(* CODESYS project Mehatronika_seminarski.project
   Title: PMS_LV9_z1
   Version: 0.0.0.0
   Author: CA Simple

Project tree, tasks and I/O mapping:
  MyController : TM238LDD24DT, Schneider Electric, order no. TM238LDD24DT, version 4.0.1.28
      settings: OpcUa Enable = False
    application Application
      task MAST (cyclic, interval 20 ms, priority 15, watchdog 100 ms x 1) calls POU
      global variables GVL
      program POU [SFC]: Init_entry, Step4_entry, kafa0_active, kafa0_entry, Step1_entry, Step2_entry, kafa0_exit, caj1_active, kafa1_exit, kafa2_active, kafa2_exit, kafa1_active, caj2_active, caj1_exit, caj2_exit, caj0_entry, caj0_exit, caj0_active, kakao0_entry, kapucino0_entry, kakao0_exit, kapucino0_exit, kakao0_active, kapucino0_active, kakao1_active, kakao1_exit, kakao2_active, kakao2_exit, kapucino1_active, kapucino1_exit, kapucino3_active, kapucino3_exit, kapucino2_active, kapucino2_exit, kafa1_entry, kafa2_entry, caj1_entry, caj2_entry, kakao1_entry, kapucino1_entry, kakao2_entry, kapucino2_entry, kapucino3_entry, Init_active, preuzimanje_active_0, Init_exit, preuzimanje_exit
      Symbols
    Embedded Functions
      IO : IO, Schneider Electric, version 4.0.1.28
          input  Application.polaKM : BOOL  // IW0.I0
          input  Application.jedanKM : BOOL  // IW0.I1
          input  Application.dvaKM : BOOL  // IW0.I2
          input  Application.kafa : BOOL  // IW0.I3
          input  Application.caj : BOOL  // IW0.I4
          input  Application.kakao : BOOL  // IW0.I5
          input  Application.kapucino : BOOL  // IW0.I6
          output Application.voda : BOOL  // QW0.Q0
          output Application.posuda1 : BOOL  // QW0.Q1
          output Application.posuda2 : BOOL  // QW0.Q2
          output Application.posuda3 : BOOL  // QW0.Q3
          output Application.posuda4 : BOOL  // QW0.Q4
          output Application.posuda5 : BOOL  // QW0.Q5
          unmapped channels: IW0, QW0
      HSC : HSC, Schneider Electric, version 4.0.1.28
      PTO_PWM : PTO_PWM, Schneider Electric, version 4.0.1.28
    Serial Line
      SoMachine_Network_Manager : SoMachine-Network Manager, Schneider Electric, version 4.0.0.2
  HMIS5T : HMIS5T, Schneider Electric, order no. HMIS5T, version 3.5.3.54
    HMI Application
    COM1
      SoMachine_Network_Manager1 : SoMachine-Network Manager, Schneider Electric, version 4.0.0.2
    Ethernet
      SoMachine_Network_Manager2 : SoMachine-Network Manager, Schneider Electric, version 4.0.0.2
    USB
      SoMachine_Network_Manager3 : SoMachine-Network Manager, Schneider Electric, version 4.0.0.2
  Vijeo Designer Project Container Data
  Vijeo Designer Project Container
*)

// MyController/Application/GVL
VAR_GLOBAL
END_VAR
VAR_GLOBAL
	petKM: BOOL;
	dvaKM: BOOL;
	jedanKM: BOOL;
	polaKM: BOOL;
	posuda5: BOOL;
	posuda4: BOOL;
	posuda3: BOOL;
	posuda2: BOOL;
	posuda1: BOOL;
	voda: BOOL;
	kapucino: BOOL;
	kakao: BOOL;
	caj: BOOL;
	kafa: BOOL;
	iznos: REAL := 0;
	kafa_iznos: BOOL;
	caj_iznos: BOOL;
	kakao_iznos: BOOL;
	kapucino_iznos: BOOL;
	kafa_gotova: BOOL;
	caj_gotov: BOOL;
	kakao_gotov: BOOL;
	kapucino_gotov: BOOL;
	kafa_u_proizvodnji: BOOL;
	caj_u_proizvodnji: BOOL;
	kakao_u_proizvodnji: BOOL;
	kapucino_u_proizvodnji: BOOL;
	proizvod_pokupljen: BOOL;
END_VAR

// MyController/Application/POU
PROGRAM POU
VAR
	okidac_posuda5: BOOL;
	okidac_posuda4: BOOL;
	okidac_posuda3: BOOL;
	okidac_posuda2: BOOL;
	okidac_posuda1: BOOL;
	okidac_voda: BOOL;
	posuda5_timer: TP;
	posuda5_f_trig: F_TRIG;
	posuda4_timer: TP;
	posuda4_f_trig: F_TRIG;
	posuda3_timer: TP;
	posuda3_f_trig: F_TRIG;
	posuda2_timer: TP;
	posuda2_f_trig: F_TRIG;
	posuda1_timer: TP;
	posuda1_f_trig: F_TRIG;
	voda_timer: TP;
	voda_f_trig: F_TRIG;
	pomocna: BOOL;
END_VAR

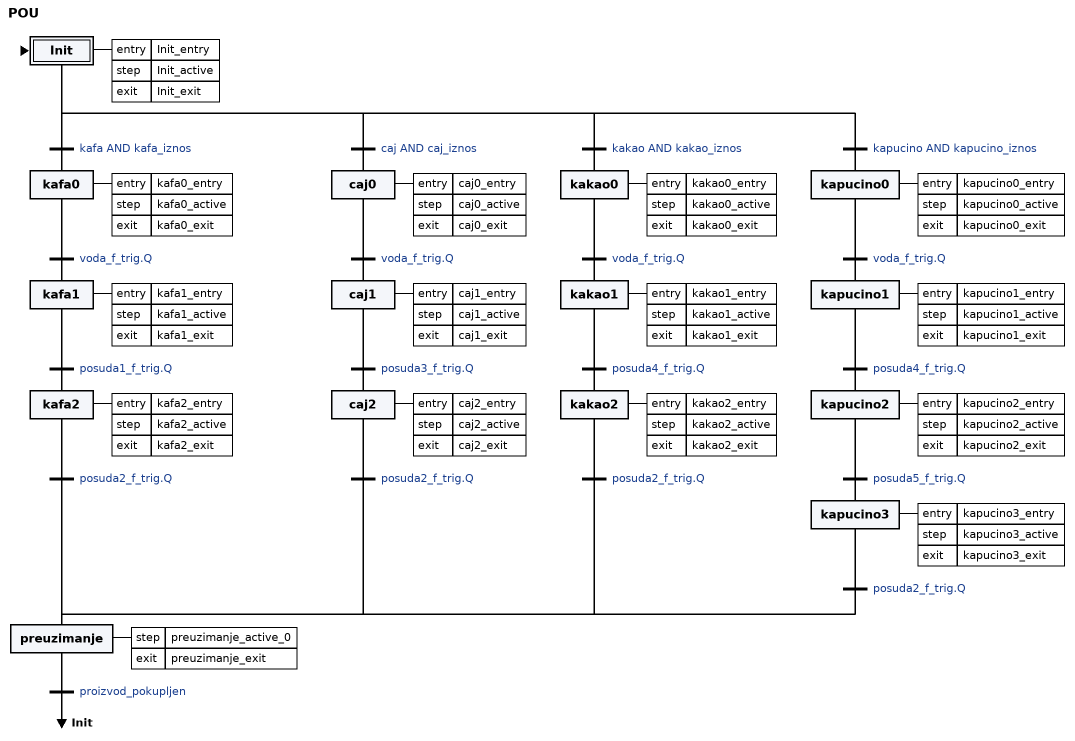
INITIAL_STEP Init:
    Init_entry(P1);  // entry action
    Init_active(N);  // step action
    Init_exit(P0);  // exit action
END_STEP
TRANSITION FROM Init TO kafa0
    := kafa AND kafa_iznos;
END_TRANSITION
STEP kafa0:
    kafa0_entry(P1);  // entry action
    kafa0_active(N);  // step action
    kafa0_exit(P0);  // exit action
END_STEP
TRANSITION FROM kafa0 TO kafa1
    := voda_f_trig.Q;
END_TRANSITION
STEP kafa1:
    kafa1_entry(P1);  // entry action
    kafa1_active(N);  // step action
    kafa1_exit(P0);  // exit action
END_STEP
TRANSITION FROM kafa1 TO kafa2
    := posuda1_f_trig.Q;
END_TRANSITION
STEP kafa2:
    kafa2_entry(P1);  // entry action
    kafa2_active(N);  // step action
    kafa2_exit(P0);  // exit action
END_STEP
TRANSITION FROM kafa2 TO preuzimanje
    := posuda2_f_trig.Q;
END_TRANSITION
TRANSITION FROM Init TO caj0
    := caj AND caj_iznos;
END_TRANSITION
STEP caj0:
    caj0_entry(P1);  // entry action
    caj0_active(N);  // step action
    caj0_exit(P0);  // exit action
END_STEP
TRANSITION FROM caj0 TO caj1
    := voda_f_trig.Q;
END_TRANSITION
STEP caj1:
    caj1_entry(P1);  // entry action
    caj1_active(N);  // step action
    caj1_exit(P0);  // exit action
END_STEP
TRANSITION FROM caj1 TO caj2
    := posuda3_f_trig.Q;
END_TRANSITION
STEP caj2:
    caj2_entry(P1);  // entry action
    caj2_active(N);  // step action
    caj2_exit(P0);  // exit action
END_STEP
TRANSITION FROM caj2 TO preuzimanje
    := posuda2_f_trig.Q;
END_TRANSITION
TRANSITION FROM Init TO kakao0
    := kakao AND kakao_iznos;
END_TRANSITION
STEP kakao0:
    kakao0_entry(P1);  // entry action
    kakao0_active(N);  // step action
    kakao0_exit(P0);  // exit action
END_STEP
TRANSITION FROM kakao0 TO kakao1
    := voda_f_trig.Q;
END_TRANSITION
STEP kakao1:
    kakao1_entry(P1);  // entry action
    kakao1_active(N);  // step action
    kakao1_exit(P0);  // exit action
END_STEP
TRANSITION FROM kakao1 TO kakao2
    := posuda4_f_trig.Q;
END_TRANSITION
STEP kakao2:
    kakao2_entry(P1);  // entry action
    kakao2_active(N);  // step action
    kakao2_exit(P0);  // exit action
END_STEP
TRANSITION FROM kakao2 TO preuzimanje
    := posuda2_f_trig.Q;
END_TRANSITION
TRANSITION FROM Init TO kapucino0
    := kapucino AND kapucino_iznos;
END_TRANSITION
STEP kapucino0:
    kapucino0_entry(P1);  // entry action
    kapucino0_active(N);  // step action
    kapucino0_exit(P0);  // exit action
END_STEP
TRANSITION FROM kapucino0 TO kapucino1
    := voda_f_trig.Q;
END_TRANSITION
STEP kapucino1:
    kapucino1_entry(P1);  // entry action
    kapucino1_active(N);  // step action
    kapucino1_exit(P0);  // exit action
END_STEP
TRANSITION FROM kapucino1 TO kapucino2
    := posuda4_f_trig.Q;
END_TRANSITION
STEP kapucino2:
    kapucino2_entry(P1);  // entry action
    kapucino2_active(N);  // step action
    kapucino2_exit(P0);  // exit action
END_STEP
TRANSITION FROM kapucino2 TO kapucino3
    := posuda5_f_trig.Q;
END_TRANSITION
STEP kapucino3:
    kapucino3_entry(P1);  // entry action
    kapucino3_active(N);  // step action
    kapucino3_exit(P0);  // exit action
END_STEP
TRANSITION FROM kapucino3 TO preuzimanje
    := posuda2_f_trig.Q;
END_TRANSITION
STEP preuzimanje:
    preuzimanje_active_0(N);  // step action
    preuzimanje_exit(P0);  // exit action
END_STEP
TRANSITION FROM preuzimanje TO Init
    := proizvod_pokupljen;
END_TRANSITION

ACTION Init_entry:

kafa_iznos := FALSE;
caj_iznos := FALSE;
kakao_iznos := FALSE;
kapucino_iznos := FALSE;

kafa_u_proizvodnji := FALSE;
caj_u_proizvodnji := FALSE;
kakao_u_proizvodnji := FALSE;
kapucino_u_proizvodnji := FALSE;

okidac_posuda1 := FALSE;
okidac_posuda2 := FALSE;
okidac_posuda3 := FALSE;
okidac_posuda4 := FALSE;
okidac_posuda5 := FALSE;
okidac_voda := FALSE;

voda_f_trig ( CLK := pomocna );
posuda1_f_trig ( CLK := pomocna );
posuda2_f_trig ( CLK := pomocna );
posuda3_f_trig ( CLK := pomocna );
posuda4_f_trig ( CLK := pomocna );
posuda5_f_trig ( CLK := pomocna );
END_ACTION

ACTION Step4_entry:
okidac_voda := TRUE;
END_ACTION

ACTION kafa0_active:
voda_timer ( IN := okidac_voda , PT:= T#5S );
voda := voda_timer.Q;



voda_f_trig (CLK:= voda_timer.Q);
okidac_voda := FALSE;
END_ACTION

ACTION kafa0_entry:
iznos := iznos -1;
kafa := FALSE;
okidac_voda := TRUE;

kafa_u_proizvodnji := TRUE;
END_ACTION

ACTION Step1_entry:
okidac_voda := TRUE;
END_ACTION

ACTION Step2_entry:
okidac_voda := TRUE;
END_ACTION

ACTION kafa0_exit:
okidac_posuda1 := TRUE;
END_ACTION

ACTION caj1_active:
posuda3_timer(IN := okidac_posuda3, PT := T#1S);
posuda3 := posuda3_timer.Q;

posuda3_f_trig (CLK := posuda3_timer.Q);
okidac_posuda3 := FALSE;
END_ACTION

ACTION kafa1_exit:
okidac_posuda1 := FALSE;
okidac_posuda2 := TRUE;
END_ACTION

ACTION kafa2_active:
posuda2_timer(IN := okidac_posuda2, PT := T#1S);
posuda2 := posuda2_timer.Q;


posuda2_f_trig (CLK := posuda2_timer.Q);
okidac_posuda2 := FALSE;
END_ACTION

ACTION kafa2_exit:
okidac_posuda2 := FALSE;
okidac_posuda3 := TRUE;

kafa_u_proizvodnji := FALSE;
kafa_gotova :=TRUE;
END_ACTION

ACTION kafa1_active:
posuda1_timer(IN := okidac_posuda1, PT := T#5S);
posuda1 := posuda1_timer.Q;



posuda1_f_trig (CLK := posuda1_timer.Q);
okidac_posuda1 := FALSE;
END_ACTION

ACTION caj2_active:
posuda2_timer(IN := okidac_posuda2, PT := T#2S);
posuda2 := posuda2_timer.Q;

okidac_posuda2 := FALSE;

posuda2_f_trig (CLK := posuda2_timer.Q);
END_ACTION

ACTION caj1_exit:

okidac_posuda2 := TRUE;
END_ACTION

ACTION caj2_exit:
okidac_posuda2 := TRUE;

caj_u_proizvodnji := FALSE;
caj_gotov :=TRUE;
END_ACTION

ACTION caj0_entry:
iznos := iznos - 0.5;
caj := FALSE;
okidac_voda := TRUE;

caj_u_proizvodnji := TRUE;
END_ACTION

ACTION caj0_exit:

okidac_posuda3 := TRUE;
END_ACTION

ACTION caj0_active:
voda_timer ( IN := okidac_voda , PT:= T#5S );
voda := voda_timer.Q;


voda_f_trig (CLK:= voda_timer.Q);
okidac_voda := FALSE;
END_ACTION

ACTION kakao0_entry:
iznos := iznos - 1;
kakao := FALSE;
okidac_voda := TRUE;

kakao_u_proizvodnji := TRUE;
END_ACTION

ACTION kapucino0_entry:
iznos := iznos - 2;
kapucino := FALSE;
okidac_voda := TRUE;

kapucino_u_proizvodnji := TRUE;
END_ACTION

ACTION kakao0_exit:
okidac_posuda4 := TRUE;
END_ACTION

ACTION kapucino0_exit:
okidac_posuda4 := TRUE;
END_ACTION

ACTION kakao0_active:
voda_timer ( IN := okidac_voda , PT:= T#5S );
voda := voda_timer.Q;

voda_f_trig (CLK:= voda_timer.Q);
okidac_voda := FALSE;
END_ACTION

ACTION kapucino0_active:
voda_timer ( IN := okidac_voda , PT:= T#5S );
voda := voda_timer.Q;



voda_f_trig (CLK:= voda_timer.Q);
okidac_voda := FALSE;
END_ACTION

ACTION kakao1_active:
posuda4_timer(IN := okidac_posuda4, PT := T#2S);
posuda4 := posuda4_timer.Q;



posuda4_f_trig (CLK := posuda4_timer.Q);
okidac_posuda4 := FALSE;
END_ACTION

ACTION kakao1_exit:
okidac_posuda4 := FALSE;
okidac_posuda2 := TRUE;
END_ACTION

ACTION kakao2_active:
posuda2_timer(IN := okidac_posuda2, PT := T#2S);
posuda2 := posuda2_timer.Q;



posuda2_f_trig (CLK := posuda2_timer.Q);
okidac_posuda2 := FALSE;
END_ACTION

ACTION kakao2_exit:
okidac_posuda2 := TRUE;

kakao_u_proizvodnji := FALSE;
kakao_gotov :=TRUE;
END_ACTION

ACTION kapucino1_active:
posuda4_timer(IN := okidac_posuda4, PT := T#2S);
posuda4 := posuda4_timer.Q;



posuda4_f_trig (CLK := posuda4_timer.Q);
okidac_posuda4 := FALSE;
END_ACTION

ACTION kapucino1_exit:
okidac_posuda4 := FALSE;
okidac_posuda5 := TRUE;
END_ACTION

ACTION kapucino3_active:
posuda2_timer(IN := okidac_posuda2, PT := T#2S);
posuda2 := posuda2_timer.Q;

posuda2_f_trig (CLK := posuda2_timer.Q);
okidac_posuda2 := FALSE;
END_ACTION

ACTION kapucino3_exit:
okidac_posuda2 := TRUE;

kapucino_u_proizvodnji := FALSE;
kapucino_gotov := TRUE;
END_ACTION

ACTION kapucino2_active:
posuda5_timer(IN := okidac_posuda5, PT := T#5S);
posuda5 := posuda5_timer.Q;



posuda5_f_trig (CLK := posuda5_timer.Q);
okidac_posuda5 := FALSE;
END_ACTION

ACTION kapucino2_exit:
okidac_posuda5 := FALSE;
okidac_posuda2 := TRUE;
END_ACTION

ACTION kafa1_entry:

END_ACTION

ACTION kafa2_entry:

END_ACTION

ACTION caj1_entry:

END_ACTION

ACTION caj2_entry:

END_ACTION

ACTION kakao1_entry:

END_ACTION

ACTION kapucino1_entry:

END_ACTION

ACTION kakao2_entry:

END_ACTION

ACTION kapucino2_entry:

END_ACTION

ACTION kapucino3_entry:

END_ACTION

ACTION Init_active:

kafa_iznos := FALSE;
caj_iznos := FALSE;
kakao_iznos := FALSE;
kapucino_iznos := FALSE;

kafa_gotova := FALSE;
caj_gotov := FALSE;
kakao_gotov := FALSE;
kapucino_gotov := FALSE;



IF ( iznos ) > 10 THEN
	
	polaKM := FALSE;
	jedanKM := FALSE;
	dvaKM := FALSE;
	petKM := FALSE;
	
	kafa_iznos := TRUE;
	caj_iznos := TRUE;
	kakao_iznos := TRUE;
	kapucino_iznos := TRUE;

ELSE
	
	IF polaKM = TRUE THEN
	iznos := iznos + 0.5; 
		polaKM := FALSE;
	END_IF;
	
	IF jedanKM = TRUE THEN
		iznos := iznos + 1;
		jedanKM := FALSE;
	END_IF;
	
	IF dvaKM = TRUE THEN
		iznos := iznos + 2;
		dvaKM := FALSE;
	END_IF;
	
	IF petKM = TRUE THEN
		iznos := iznos + 5;
		petKM := FALSE;
	END_IF;
	
	IF iznos >= 0.5 THEN
		caj_iznos := TRUE;
	END_IF;
	
	IF iznos >= 1 THEN
		kafa_iznos := TRUE;
		kakao_iznos := TRUE;
	END_IF;
	
	IF iznos >= 2 THEN
		kapucino_iznos := TRUE;
	END_IF;

END_IF;
END_ACTION

ACTION preuzimanje_active_0:

END_ACTION

ACTION Init_exit:
proizvod_pokupljen := FALSE;
END_ACTION

ACTION preuzimanje_exit:
iznos := 0;
END_ACTION

END_PROGRAM
